Universal Robots PolyScope program: 202505241409.urp

Program 202505241409 (installation=20240827 directory=/programs/collection createdIn=5.15.1 lastSavedIn=5.15.1 robotSerialNumber=20245500285)
Calibrated DH parameters: a=[0.000097, -0.210459, -0.026602, 0.000137, 0.000078, 0]; d=[0.162601, 254.180657, -54.076236, -199.970743, 0.099615, 0.099684]; alpha=[1.569796, -0.001455, 0.001957, 1.570525, -1.571561, 0]; deltaTheta=[0, -1.053331, 8.839472, -1.50296, 0.000002, 0]
InitVariablesNode
Robot Program (runOnlyOnce=false)
  mode := 2
  '0-空闲/1-基础验证/2-中心点Z/3-全点Z'
  step_x := 0.004
  step_y := 0.004
  step_z := 0.0002
  step_tcp := 0.0001
  var_x := [0,-1,1,-1,1,0]
  var_y := [0,-1,1,1,-1,0]
  '一维路点(0,0)(-1,1)(1,1)(-1,-1)(1,-1)'
  '默认一维路点(0,0)'
  Script: start0 = rpc_factory("xmlrpc","http://192.168.1.7:9125/RPC2")
  SuppressedNode
    Script: soket_open("192.168.1.7",9126)
  Popup Message (haltProgram=false inputType=Variable) variable=mode
  MoveJ speed 60 deg/s, acceleration 80 deg/s^2 (useActiveTCP=true) feature=Base
    Waypoint 路点_1: TCP in base x=804.437 y=122.593 z=257.99 mm, rx=1.21 ry=1.2108 rz=1.2121 rad; joints [178.627, -48.174, 103.133, -234.956, -88.629, 180.007] deg; TCP offset x=-0.17 y=0 z=192.95 mm, rx=0 ry=0 rz=0 rad
    '过渡点'
    Waypoint tcp: TCP in base x=804.418 y=122.593 z=253.777 mm, rx=1.2099 ry=1.2108 rz=1.2121 rad; joints [178.627, -47.696, 103.127, -235.429, -88.629, 180.004] deg
    '受力0，距离0'
  If mode==0
    Popup Message (haltProgram=false message=空闲模式 inputType=Text)
    SuppressedNode
      Script: start0.trigger_s_key()
    SuppressedNode
      Wait Sleep waitTime=7
  ElseIf mode==1
    Popup Message (haltProgram=false message=基础TCP位置验证 inputType=Text)
    step := 0
    Loop Counting (count=20) loopVariable(name=循环_1)
      step := step+1
      tcptcp := pose_add(tcp, p[0,0,-step_tcp*step,0,0,0])
      tcptcpz := tcptcp[2]
      Popup Message (haltProgram=false inputType=Variable) variable=tcptcpz
      SuppressedNode
        Script: socket_open("192.168.1.7",9126)
      SuppressedNode
        Script: socket_send("123")
      SuppressedNode
        Script: socket_close()
      MoveJ speed 60 deg/s, acceleration 80 deg/s^2 (useActiveTCP=true) feature=Base
        Popup Message (haltProgram=false inputType=Variable) variable(name=tcptcp)
        Waypoint Variable (Variable): variable=tcptcp
      SuppressedNode
        Script: start0.send_float_data(tcptcpz)
      SuppressedNode
        Script: start0.trigger_s_key()
      SuppressedNode
        Wait Sleep waitTime=7
    Popup Message (haltProgram=false message=基础TCP位置验证 inputType=Text)
  ElseIf mode==2
    Popup Message (haltProgram=false message=中心点Z方向测试 inputType=Text)
    step := 0
    Loop Counting (count=25) loopVariable(name=循环_2)
      step := step+1
      tcptcp := pose_add(tcp, p[0,0,-step*step_z,0,0,0])
      Popup Message (haltProgram=false inputType=Variable) variable=step
      MoveJ speed 60 deg/s, acceleration 80 deg/s^2 (useActiveTCP=true) feature=Base
        Popup Message (haltProgram=false inputType=Variable) variable=tcptcp
        Waypoint Variable (Variable): variable=tcptcp
      var_1 := tcptcp[0]
      var_2 := tcptcp[1]
      var_3 := tcptcp[2]
      SuppressedNode
        Popup Message (haltProgram=false message=andand inputType=Text)
      Script: start0.xyz_s(var_1,var_2,var_3)
      SuppressedNode
        Script: start0.trigger_and_send_xyz(var_1,var_2,var_3)
      SuppressedNode
        Popup Message (haltProgram=false message=xyz s inputType=Text)
      SuppressedNode
        Script: start0.send_xyz_coordinates(var_1,var_2,var_3)
      SuppressedNode
        Wait Sleep waitTime=7
      SuppressedNode
        Script: start0.trigger_s_key()
      Wait Sleep waitTime=7
    Popup Message (haltProgram=false message=中心点Z方向测试 inputType=Text)
  ElseIf mode==22
    Popup Message (haltProgram=false message=中心点Z方向测试 inputType=Text)
    step := 0
    Loop Counting (count=25) loopVariable(name=循环_3)
      step := step+1
      tcptcp := pose_add(tcp, p[0,0,-step*step_z,0,0,0])
      SuppressedNode
        Popup Message (haltProgram=false inputType=Variable) variable=step
      MoveJ speed 60 deg/s, acceleration 80 deg/s^2 (useActiveTCP=true) feature=Base
        SuppressedNode
          Popup Message (haltProgram=false inputType=Variable) variable=tcptcp
        Waypoint Variable (Variable): variable=tcptcp
      var_1 := tcptcp[0]
      var_2 := tcptcp[1]
      var_3 := tcptcp[2]
      Script: start0.send_xyz_coordinates(var_1,var_2,var_3)
      Wait Sleep waitTime=1
      Script: start0.trigger_s_key()
      Wait Sleep waitTime=7
    Popup Message (haltProgram=false message=中心点Z方向测试 inputType=Text)
  ElseIf mode==3
    Popup Message (haltProgram=false message=全点Z测试 inputType=Text)
    xy := 0
    Loop Counting (count=5) loopVariable(name=循环_4)
      MoveJ speed 60 deg/s, acceleration 80 deg/s^2 (useActiveTCP=true) feature=Base
        Waypoint 路点_1: TCP in base x=804.437 y=122.593 z=257.99 mm, rx=1.21 ry=1.2108 rz=1.2121 rad; joints [178.627, -48.174, 103.133, -234.956, -88.629, 180.007] deg
      xy := xy+1
      step := 0
      Loop Counting (count=25) loopVariable(name=循环_5)
        step := step+1
        tcptcp := pose_add(tcp, p[step_x*var_x[xy],step_y*var_y[xy],-step*step_z,0,0,0])
        MoveJ speed 60 deg/s, acceleration 80 deg/s^2 (useActiveTCP=true) feature=Base
          Popup Message (haltProgram=false inputType=Variable) variable=tcptcp
          Waypoint Variable (Variable): variable=tcptcp
        Script: start0.trigger_s_key()
        Wait Sleep waitTime=7
    Popup Message (haltProgram=false message=全点Z测试 inputType=Text)
  ElseIf mode==33
    Popup Message (haltProgram=false message=全点Z测试 inputType=Text)
    xy := 0
    Loop Counting (count=5) loopVariable(name=循环_6)
      MoveJ speed 60 deg/s, acceleration 80 deg/s^2 (useActiveTCP=true) feature=Base
        Waypoint 路点_1: TCP in base x=804.437 y=122.593 z=257.99 mm, rx=1.21 ry=1.2108 rz=1.2121 rad; joints [178.627, -48.174, 103.133, -234.956, -88.629, 180.007] deg
      xy := xy+1
      step := 0
      Loop Counting (count=25) loopVariable(name=循环_7)
        step := step+1
        tcptcp := pose_add(tcp, p[step_x*var_x[xy],step_y*var_y[xy],-step*step_z,0,0,0])
        MoveJ speed 60 deg/s, acceleration 80 deg/s^2 (useActiveTCP=true) feature=Base
          SuppressedNode
            Popup Message (haltProgram=false inputType=Variable) variable=tcptcp
          Waypoint Variable (Variable): variable=tcptcp
        Wait Sleep waitTime=1
        Script: start0.trigger_s_key()
        Wait Sleep waitTime=7
    Popup Message (haltProgram=false message=全点Z测试 inputType=Text)
